{attribute 'qualified_only'}
{attribute 'strict'}
TYPE E_PvSource :
(
    PV1 := 0,
    PV2 := 1
);
END_TYPE

(* stored: Version 1.1.0.1, ProductVersion 3.1.4026.12
   DUT E_PvSource: Id {028cb00b-ab69-4a3f-bb06-6a0e8fd8d4f0} *)
